{attribute 'qualified_only'}
{attribute 'strict'}
TYPE EControlModeSmd12 :
(
	CurrentMode, 
	PowerMode
);
END_TYPE

(* stored: Version 1.1.0.1, ProductVersion 3.1.4024.3
   DUT EControlModeSmd12: Id {1b743453-1177-4400-a157-f3d1e796c610} *)
